INTERFACE I_PackML_BaseModule EXTENDS I_CyclicFB, I_PackML_Control

PROPERTY CurrentAlarmSeverity : TcEventSeverity
GET
END_GET
END_PROPERTY

PROPERTY LogModeChanges : BOOL
GET
END_GET
SET
END_SET
END_PROPERTY

PROPERTY LogStateChanges : BOOL
GET
END_GET
SET
END_SET
END_PROPERTY

PROPERTY Name : STRING
GET
END_GET
SET
END_SET
END_PROPERTY

PROPERTY ParentResponseDefinitions : ARRAY[0..4] OF E_AlarmResponse
GET
END_GET
SET
END_SET
END_PROPERTY

END_INTERFACE

(* stored: Version 1.1.0.1, ProductVersion 3.1.4024.12
   Itf I_PackML_BaseModule: Id {eca4a56b-850e-483e-b687-2de3b3950c24}
   Property CurrentAlarmSeverity: Id {6330edd2-66f0-4e35-86ff-3d09385aa422}
   Get Get: Id {2352a7a5-1a04-4154-bd74-fbb96f906eec}
   Property LogModeChanges: Id {3ebf3a99-dead-418c-b471-054c7c8d6544}
   Get Get: Id {e04dfd29-bd9f-4f54-828e-2fc4045c23bc}
   Set Set: Id {1785a2f9-a528-437d-84c4-405797055f1f}
   Property LogStateChanges: Id {1b008608-b316-4d3a-ba87-f437076859ca}
   Get Get: Id {66bc6c53-f9e2-4511-89b6-29fb383f77e7}
   Set Set: Id {a9b78c0c-4b3e-4169-a6c7-77bf1bd91d29}
   Property Name: Id {da8f2502-5e83-49c9-bcb7-07c02f3fcb7b}
   Get Get: Id {c93e64d6-b7f5-4fa1-96b7-7e8cdadc8f67}
   Set Set: Id {0e6ed32b-5954-42fd-b96a-59359710d227}
   Property ParentResponseDefinitions: Id {e3645d3e-2142-4d00-bb59-0dedc9223132}
   Get Get: Id {20c65c99-40c2-4b98-8141-816006beb6ed}
   Set Set: Id {ae399fa5-e93f-4526-82f5-2b92335ced38} *)
